INTERFACE I_V1_VirtualInputSource EXTENDS I_VirtualInputSource

PROPERTY nV1_TimeLine : ULINT
GET
END_GET
END_PROPERTY

PROPERTY bV1_bProductionMode : BOOL
GET
END_GET
END_PROPERTY

PROPERTY nV1_lScheduledTime : LINT
GET
END_GET
END_PROPERTY

PROPERTY nV1_uDefectiveCount : ULINT
GET
END_GET
END_PROPERTY

PROPERTY nV1_lStartTime : LWORD
GET
END_GET
END_PROPERTY

PROPERTY nV1_lStopTime : LWORD
GET
END_GET
END_PROPERTY

PROPERTY bV1_bConfigure : BOOL
GET
END_GET
END_PROPERTY

PROPERTY bV1_bReset : BOOL
GET
END_GET
END_PROPERTY

PROPERTY bV1_bTest : BOOL
GET
END_GET
END_PROPERTY

PROPERTY nV1_uTotalCount : ULINT
GET
END_GET
END_PROPERTY

END_INTERFACE

(* stored: Itf I_V1_VirtualInputSource: Id 9077eff0-1e38-4d28-a561-eca7188a3413
   Property nV1_TimeLine: Id d6a89746-74a2-4baf-93ee-50e8c0ecde3b
   Get Get: Id 32385617-aaa0-410c-bceb-c44d89695eba
   Property bV1_bProductionMode: Id 34fbf626-267c-4d48-84de-ab048657b8ab
   Get Get: Id dfb288e1-9c45-4adf-9053-cbf217a80dd5
   Property nV1_lScheduledTime: Id a9aef586-a9f5-4419-8170-bf6fc7018bec
   Get Get: Id dcb7d244-0ae0-480b-ab23-b11842d37402
   Property nV1_uDefectiveCount: Id 2dbed273-b49e-47ee-b117-ed34f105f8f5
   Get Get: Id 5497485c-ab2e-4cde-814f-5fde0a6615e5
   Property nV1_lStartTime: Id 4f505f8a-338d-4c94-9829-5e4d0de584ef
   Get Get: Id e0ca0f2b-eab2-4114-9ec6-78be6a0da8dd
   Property nV1_lStopTime: Id ce130914-5eba-40e3-aeb4-d0872295c74e
   Get Get: Id 6bde8e15-c95a-416e-8e7f-2d1a859bfdcf
   Property bV1_bConfigure: Id fd0632c8-331f-44d3-80fd-d4772471e871
   Get Get: Id e0644c3f-6742-420f-a83c-1414f91effcf
   Property bV1_bReset: Id 8c86cd09-5c9e-4044-b29d-8fec6025f93f
   Get Get: Id 3726bf81-eaba-478b-8802-a6db77068d7a
   Property bV1_bTest: Id 0ba4d291-1878-4c10-8cd1-030b4ee15494
   Get Get: Id c7ec5049-2ce3-402f-83a4-3cead518a09f
   Property nV1_uTotalCount: Id 75c1ddc5-6ba0-4608-a367-8da1cd4ac92b
   Get Get: Id 8c8e9150-4ad2-41a3-b88a-e1b80e96876f *)
